PROGRAM PILS_DEVICES
VAR
END_VAR

//Interface between PILS and TwinCAT variables
//Example code of how to link the varaibles and PILS:
(*
fbMotorM1(stAxisStruct:= astAxes[1], stDeviceStructPILS:= stMotorM1, stAxisPar:= stMotorM1Param);
stMotor1Temp.fValue := Axis_1.fMotTemp1;
stMotorM1EncoderRaw.nValue := nEncoderValueAxis1;
fbPneumaticP1(stPneumaticStruct:= astPneumaticAxes[1], stDeviceStructPILS:= stPneumaticP1);

//Cabinet Monitoring
actMonitoring();

//Pressure sensors limits
actPressureSensors();

//PTP
actPTP();
*)

ACTION actMonitoring:
(*IF (Cabinet_Monitoring.fbCabinetMonitoring.nAlarmGrpBitNumber AND 16#00104F) <> 0 THEN
    stCabinetStatus.nStatus := E_Statusword32AlarmState.eStatuswordAlarmStateErrorHw;
ELSIF (Cabinet_Monitoring.fbCabinetMonitoring.nAlarmGrpBitNumber AND 16#000730) <> 0 THEN
    stCabinetStatus.nStatus := E_Statusword32AlarmState.eStatuswordAlarmStateWarningHi;
ELSIF (Cabinet_Monitoring.fbCabinetMonitoring.nAlarmGrpBitNumber AND 16#000880) <> 0 THEN
    stCabinetStatus.nStatus := E_Statusword32AlarmState.eStatuswordAlarmStateWarningLo;
ELSE
    stCabinetStatus.nStatus := E_Statusword32AlarmState.eStatuswordAlarmStateNoAlarm;
END_IF

stCabinetStatus.nStatus.0 := Cabinet_Monitoring.fbCabinetMonitoring.nAlarmGrpBitNumber.0; //HW alarm
stCabinetStatus.nStatus.1 := Cabinet_Monitoring.fbCabinetMonitoring.nAlarmGrpBitNumber.1; //HW alarm
stCabinetStatus.nStatus.2 := Cabinet_Monitoring.fbCabinetMonitoring.nAlarmGrpBitNumber.2; //HW alarm
stCabinetStatus.nStatus.3 := Cabinet_Monitoring.fbCabinetMonitoring.nAlarmGrpBitNumber.3; //HW alarm
stCabinetStatus.nStatus.4 := Cabinet_Monitoring.fbCabinetMonitoring.nAlarmGrpBitNumber.4; //Warning High
stCabinetStatus.nStatus.5 := Cabinet_Monitoring.fbCabinetMonitoring.nAlarmGrpBitNumber.5; //Warning High
stCabinetStatus.nStatus.6 := Cabinet_Monitoring.fbCabinetMonitoring.nAlarmGrpBitNumber.6; //HW alarm
stCabinetStatus.nStatus.7 := Cabinet_Monitoring.fbCabinetMonitoring.nAlarmGrpBitNumber.7; //Warning Low
stCabinetStatus.nStatus.8 := Cabinet_Monitoring.fbCabinetMonitoring.nAlarmGrpBitNumber.8; //Warning High
stCabinetStatus.nStatus.9 := Cabinet_Monitoring.fbCabinetMonitoring.nAlarmGrpBitNumber.9; //Warning High
stCabinetStatus.nStatus.10 := Cabinet_Monitoring.fbCabinetMonitoring.nAlarmGrpBitNumber.10; //Warning High
stCabinetStatus.nStatus.11 := Cabinet_Monitoring.fbCabinetMonitoring.nAlarmGrpBitNumber.11; //Warning Low
stCabinetStatus.nStatus.12 := Cabinet_Monitoring.fbCabinetMonitoring.nAlarmGrpBitNumber.12; //HW alarm
*)
END_ACTION

ACTION actPressureSensors:
(*//Pressure sensor group1
stPressureSensor1.fValue := Pneumatic_Box.fScaledAirPressureGroup1;
IF NOT Pneumatic_Box.bAirPressureLowGrp1 AND NOT Pneumatic_Box.bAirPressureHighGrp1 THEN
    stPressureSensor1.nStatus := E_Statusword32AlarmState.eStatuswordAlarmStateNoAlarm;
ELSIF Pneumatic_Box.bAirPressureLowGrp1 THEN
    stPressureSensor1.nStatus := E_Statusword32AlarmState.eStatuswordAlarmStateWarningLo;
ELSIF Pneumatic_Box.bAirPressureHighGrp1 THEN
    stPressureSensor1.nStatus := E_Statusword32AlarmState.eStatuswordAlarmStateWarningHi;
END_IF
//Pressure sensor group 2
stPressureSensor2.fValue := Pneumatic_Box.fScaledAirPressureGroup2;
IF NOT Pneumatic_Box.bAirPressureLowGrp2 AND NOT Pneumatic_Box.bAirPressureHighGrp2 THEN
    stPressureSensor2.nStatus := E_Statusword32AlarmState.eStatuswordAlarmStateNoAlarm;
ELSIF Pneumatic_Box.bAirPressureLowGrp2 THEN
    stPressureSensor2.nStatus := E_Statusword32AlarmState.eStatuswordAlarmStateWarningLo;
ELSIF Pneumatic_Box.bAirPressureHighGrp2 THEN
    stPressureSensor2.nStatus := E_Statusword32AlarmState.eStatuswordAlarmStateWarningHi;
END_IF
*)
END_ACTION

ACTION actPTP:
(*IF PILSv2.bPILSV2isInitialized THEN
    GVL_PILS.stPTPState.nValue        := SEL(EL6688_PTP.bExternalDeviceNotConnected, EL6688_PTP.nPtpState, -2);
    GVL_PILS.stPTPState.nStatus       := SEL(EL6688_PTP.fbRdRdEL6688Diag.bError OR EL6688_PTP.bExternalDeviceNotConnected,
                                             E_Statusword32AlarmState.eStatuswordAlarmStateNoAlarm,
                                             E_Statusword32AlarmState.eStatuswordAlarmStateErrorHw);
    GVL_PILS.stPTPOffset.nValue       := EL6688_PTP.nPTPOffset;
    IF EL6688_PTP.fbRdRdEL6688Diag.bError OR EL6688_PTP.bExternalDeviceNotConnected THEN
        GVL_PILS.stPTPOffset.nStatus := E_Statusword32AlarmState.eStatuswordAlarmStateErrorHw;
    ELSIF EL6688_PTP.nPTPOffset > EL6688_PTP.nSyncWindow THEN
        GVL_PILS.stPTPOffset.nStatus := E_Statusword32AlarmState.eStatuswordAlarmStateWarningHi;
    ELSIF EL6688_PTP.nPTPOffset < 0 - EL6688_PTP.nSyncWindow THEN
        GVL_PILS.stPTPOffset.nStatus := E_Statusword32AlarmState.eStatuswordAlarmStateWarningLo;
    ELSE
        GVL_PILS.stPTPOffset.nStatus  := E_Statusword32AlarmState.eStatuswordAlarmStateNoAlarm;
    END_IF
    GVL_PILS.stPTPSyncSeqNum.nValue   := UINT_TO_INT(INT_TO_UINT(EL6688_PTP.nPtpSyncSeqNum) AND 7); // Just see if it is counting
    GVL_PILS.stPTPErrorStatus.nValue  := UDINT_TO_DINT(EL6688_PTP.nPTPErrorStatusBits  AND 16#0FFFFFFF);
    GVL_PILS.stPTPErrorStatus.nStatus := EL6688_PTP.nPTPErrorStatusBits;
    GVL_PILS.stPTPDcToExtTimeOffsetSystem.nValue := EL6688_PTP.nDcToExtTimeOffset;
    GVL_PILS.stDcTime64.nValue      := EL6688_PTP.nDcTime64;
    GVL_PILS.stSystemUTCtime.nValue := EL6688_PTP.nSystemUTCtime;
END_IF
*)
END_ACTION

END_PROGRAM

(* stored: Version 1.1.0.1
   POU PILS_DEVICES: Id {c13d0ec1-dadc-4beb-a3f1-3a752770c4f8}, SpecialFunc None
   Action actMonitoring: Id {93519f21-7373-0d3a-1d58-f89b51f7b818}
   Action actPressureSensors: Id {0da25c4d-63ff-0502-1976-f9d8e0c61ba8}
   Action actPTP: Id {b4bb5444-1083-09ad-366e-a71a22299f4b} *)
